(* IEC 61131-3 sources: ae-debugging/src/fbProgram, 2 files *)

(* ---- fb.st ---- *)
FUNCTION_BLOCK Fb
    VAR_EXTERNAL
        UpCounterInt : INT;
    END_VAR
    VAR
        static : INT;
    END_VAR
    VAR_TEMP
        temp : INT;
    END_VAR
    VAR_OUTPUT
        returnValue : INT;
    END_VAR

    static := UpCounterInt MOD 7;
    temp := 42;

    IF static = 0 THEN
        temp := 1337;
    END_IF;

    returnValue := temp;
END_FUNCTION_BLOCK

(* ---- fbProgram.st ---- *)
PROGRAM FbProgram
    VAR_EXTERNAL
        UpCounterInt : INT;
    END_VAR

    VAR
        functionBlock : Fb;
    END_VAR

    UpCounterInt := UpCounterInt + 1;

    functionBlock();

END_PROGRAM
